(* CODESYS project GenPanel.project

Project tree, tasks and I/O mapping:
  Device : SPK1xx, Production association OWEN, version 3.5.4.26
    application Application
      libraries: Standard, * (System); SysCom, 3.5.5.0 (System); Memory, 3.5.7.0 (3S - Smart Software Solutions GmbH); CmpVisuHandler, 3.5.11.0 (System); SysTypes Interfaces, * (System); VisuDialogs, * (System)
      task MainTask (cyclic, interval t#500ms, priority 1) calls PLC_PRG
      task Task_ReadMercury230 (cyclic, interval t#1ms, priority 20) calls POU_ReadPortGen, POU_VisuDailyEnergies
      task VISU_TASK (cyclic, interval 150 ms, priority 6) calls VisuElems.Visu_Prg
      task Task_DispatchDevices (cyclic, interval t#600ms, priority 20) calls POU_DispatchDevices
      task Task_TraceCurrents (cyclic, interval t#150ms, priority 31) calls POU_TraceCurrents
      task Task_Vis_P (cyclic, interval t#100ms, priority 5) calls POU_TracePowerActive
      task Task_WriteFile (cyclic, interval t#90ms, priority 3) calls POU_File
      task AlarmManagerTask (cyclic, interval 50 ms, priority 0) calls AlarmManager.Alarm_Prg
      program PLC_PRG [ST]
      visualisation Visualization
      visualisation Visualization_DispatchDevices
      visualisation Visualization_DailyEnergies
      visualisation Visualization_P
      global variables GVL
      visualisation Visualization_Energies
      visualisation Visualization_EnergiesDay
      data type FileWork
      visualisation Visualization_ConfigDailyView
      visualisation Visualization_Status
      Alarm Configuration
        alarm class Error (priority 10, acknowledge REP_ACK)
        alarm class Warning (priority 30, acknowledge REP)
        alarm class Info (priority 100, acknowledge REP)
        AlarmStorage
        text list AlarmGroup
        alarm group AlarmGroup
    Buzzer : Buzzer, Production association OWEN, version 3.5.4.0
        unmapped channels: Buzzer enabled, Enable buzzer
    Drives : Drives, Production association OWEN, version 3.5.4.3
        input  Application.fDebugSystem1 : BIT  // Drives info
        output Application.POU_File.fMMCMounted : BIT  // MMC Mounted
        output Application.POU_File.lwMMCSize : LWORD  // MMC size
        output Application.POU_File.lwMMCUsed : LWORD  // MMC used
        output Application.POU_File.lwMMCFree : LWORD  // MMC free
        unmapped channels: FS size, FS used, FS free, USB1 Mounted, USB1 Unmount, USB1 Unmount done, USB1 size, USB1 used, USB1 free, MMC Unmount, MMC Unmount done
    Screen : Screen, Production association OWEN, version 3.5.4.1
        unmapped channels: Get brightness, Dim time, Off time, Full brightness, Dim brightness, Off brightness, Dim visu name, Off visu name, On visu name, Wake up
    Debug : Debug, Production association OWEN, version 3.5.7.10
        input  Application.fDebugSystem : BIT  // Debug info
        input  Application.timeDebugSystem : WORD  // Debug pause
        unmapped channels: RAM used, RAM free, Open files, Processor usage, Core temp
    Modbus_COM : Modbus COM, 3S - Smart Software Solutions GmbH, version 3.4.0.0
        settings: ComPort = 2
      Modbus_Master_COM_Port : Modbus Master, COM Port, 3S - Smart Software Solutions GmbH, version 3.5.5.0
        Modbus_Slave_COM_Port : Modbus Slave, COM Port, 3S - Smart Software Solutions GmbH, version 3.5.4.0
            settings: Channel 0.Function Code = 3; Channel 0.Read Offset = 16#0001; Channel 0.Read Length = 2; Channel 0.Write Offset = 0; Channel 0.Write Length = 0; Channel 0.Cycle Time = 100; Channel 1.Function Code = 3; Channel 1.Read Offset = 16#0003; Channel 1.Read Length = 2; Channel 1.Write Offset = 0; Channel 1.Write Length = 0; Channel 1.Cycle Time = 100; Channel 2.Function Code = 3; Channel 2.Read Offset = 16#0005; Channel 2.Read Length = 2; Channel 2.Write Offset = 0; Channel 2.Write Length = 0; Channel 2.Cycle Time = 100; Channel 3.Function Code = 4; Channel 3.Read Offset = 16#0019; Channel 3.Read Length = 2; Channel 3.Write Offset = 0; Channel 3.Write Length = 0; Channel 3.Cycle Time = 100; Channel 4.Function Code = 3; Channel 4.Read Offset = 16#001B; Channel 4.Read Length = 2; Channel 4.Write Offset = 0; Channel 4.Write Length = 0; Channel 4.Cycle Time = 100; Channel 5.Function Code = 3; Channel 5.Read Offset = 16#001D; Channel 5.Read Length = 2; Channel 5.Write Offset = 0; Channel 5.Write Length = 0; Channel 5.Cycle Time = 100; Channel 6.Function Code = 3; Channel 6.Read Offset = 16#001F; Channel 6.Read Length = 2; Channel 6.Write Offset = 0;
              Channel 6.Write Length = 0; Channel 6.Cycle Time = 100; Channel 7.Function Code = 3; Channel 7.Read Offset = 16#002F; Channel 7.Read Length = 2; Channel 7.Write Offset = 0; Channel 7.Write Length = 0; Channel 7.Cycle Time = 100; Channel 8.Function Code = 3; Channel 8.Read Offset = 16#0037; Channel 8.Read Length = 2; Channel 8.Write Offset = 0; Channel 8.Write Length = 0; Channel 8.Cycle Time = 100; Channel 9.Function Code = 3; Channel 9.Read Offset = 16#00B9; Channel 9.Read Length = 1; Channel 9.Write Offset = 0; Channel 9.Write Length = 0; Channel 9.Cycle Time = 100
            input  Application.IrmsA : ARRAY[0..1] OF WORD  // Channel 0
            input  Application.IrmsB : ARRAY[0..1] OF WORD  // Channel 1
            input  Application.IrmsC : ARRAY[0..1] OF WORD  // Channel 2
            input  Application.P_A : ARRAY[0..1] OF WORD  // Channel 3
            input  Application.P_B : ARRAY[0..1] OF WORD  // Channel 4
            input  Application.P_C : ARRAY[0..1] OF WORD  // Channel 5
            input  Application.P_ABC : ARRAY[0..1] OF WORD  // Channel 6
            input  Application.S_ABC : ARRAY[0..1] OF WORD  // Channel 7
            input  Application.PF_ABCS : ARRAY[0..1] OF WORD  // Channel 8
            unmapped channels: Channel 9
  libraries: VisuSymbols, 3.5.10.0 (System); BASIC, 3.3.3.0 (OSCAT); CAA File, 3.5.3.0 (CAA Technical Workgroup)
  program POU_ReadPortGen [ST]
  program POU_DispatchDevices [ST]
  program POU_TraceCurrents [ST]
  program POU_TracePowerActive [ST]
  program POU_VisuDailyEnergies [ST]
  text list GlobalTextList
  function KAV_HEX_TO_BYTE [ST]
  program POU_File [ST]
  text list System
  image pool ImagePool
  5ce3da45-db07-42e7-a21c-a00fff4ed8f6|D:\A_Kudryashov\Documents\Мои рисунки\setup-clipart-wrench-outline-icon-clip-art_f_85-85.jpg
  Functions/
    function HEXb_TO_byteb [ST]
    function CalcCRC [ST]
    function DWORD_TO_HEXStr [ST]
*)

// Device/Application/FileWork
{attribute 'qualified_only'}
{attribute 'strict'}
TYPE FileWork :
(
	OPEN 			:= 	0,
	CREATE  		:=  10,
	READ			:=	20,
	SET_READ_POS 	:=  30,
	WRITE			:=	40,
	FLUSH			:=	50,
	CLOSE			:= 	60,
	GET_SIZE		:=	70,
	SET_POS			:=	80,
	READ_BLOCK		:=	90
);
END_TYPE

// Device/Application/GVL
VAR_GLOBAL
	IrmsA:REAL;
	IrmsB:REAL;
	IrmsC:REAL;
	Sec:BYTE;
	F_ABCS:REAL;
	PF_ABCS:real; //считанный коэф мощности
	
	P_ABCS_T:REAL;
	
	P_A:REAL; //акивна мощность фазы А
	P_B:REAL; //акивна мощность фазы B
	P_C:REAL; //акивна мощность фазы C
	P_ABC:REAL; // активная мощность
	Pq_ABC:REAL; //актвная мощость в кВт
	S_ABC:REAL; //полная мощность по фазам

	
	StartTrace:BOOL := TRUE;	//Разрешить запуск трассировки
	StopTrace:BOOL	:= FALSE;
	
	MercurySec: BYTE;  //Секунды, считанные из Меркурий230
	MercuryMin: BYTE;
	MercuryHour: BYTE;
	MercuryDay: BYTE;
	MercuryMonth: BYTE;
	MercuryYear: BYTE;
	MercuryEnergyA:DWORD;
	RealDaylyEnergyA:REAL;	//Расчитанная активная энергия за сутки 
	RealDaylyEnergyR:REAL;	//Расчитанная реактивная энергия за сутки
	RealMonthEnergyA:REAL;	//Расчитанная активная энергия за месяц
	RealMonthEnergyR:REAL;  //Расчитанная реактивная энергия за месяц             
	
	fStartTimerOpenSection: BOOL := TRUE; // Старт таймера для открытия сессии
	fStartTimerReadOpenSection:BOOL;
	fStartTimerReadTime:BOOL;
	fStartTimerReadEnergies:BOOL;
	
	DailyEnergies: ARRAY [0..24] OF REAL;
	strDailyEnergies: ARRAY [1..24] OF STRING;
	
	fFirstStartLoadDataFromFile:BOOL := true; //
	
	ReadPosition: DWORD := 5;
	fContinueRead: BOOL := FALSE; // дополнительная переменная, использования при считывании из файла
	
	fDebugSystem:BOOL := TRUE; //разрешить сбор отладочной инфы с панели
	fDebugSystem1:BOOL := TRUE; //разрешить сбор отладочной инфы с панели	
	timeDebugSystem:WORD := 5;
	
	(*
		Переменные для менеджера тревог
	*)
	fLowStorageMem:bool:=false; // используется для фиксации момента, когда на SD-карте останется меньше 20Мб
END_VAR

// Device/Application/PLC_PRG
PROGRAM PLC_PRG
VAR
	
	
END_VAR

VAR_INPUT     
	XCoord:array [0..24] of int; //координаты Х, используемые для расстановки значений мощностей по шкале
    DotY: ARRAY [1..24] OF INT; //координаты часовых точек на графике	
	DotX: ARRAY [1..24] OF INT; // координаты часовых меток на оси Y
	arrMetkaX: ARRAY [1..24] OF STRING := ['01','02','03','04','05','06','07','08','09','10','11','12','13','14','15','16','17','18','19','20','21','22','23','00']; //метки по оси Х
	
	iVar: BYTE := 16#5F;
	CRC:WORD;
	READ_ENERGIES_NOVEMBER:STRING(6) := '$5f$05$3b$00';
	l:byte;
END_VAR

l := 1;
CRC :=MEM.CRC16_Modbus(pMemoryBlock:= adr(READ_ENERGIES_NOVEMBER), uiLength:= 4);

END_PROGRAM

// POU_ReadPortGen
// This example shows how to communicate via the library SysCom.
PROGRAM POU_ReadPortGen
VAR CONSTANT
	n: BYTE := 11;
	TEST_NET: WORD := 16#5F00;
	
	AdrMercury230:string := '$5f'; // адрес текущего счетчика в формате HEX
	PURE_OPEN_CHANEL: STRING(3):= '$05$3b$00'; //команда счетчику на открытие сессии
	READ_ENERGIES_DAYLY:STRING(6) := '$5f$05$4b$00$34$C1'; //чтение потребленных энергий за сутки
	READ_ENERGIES_NOVEMBER:STRING(6) := '$5f$05$3b$00$11$01';
	OPEN_CHANEL: STRING(11) := '$5F$01$02$02$02$02$02$02$02$0D$F4';
	READ_CURRENT_TIME : STRING(6) := '$5F$04$00$43$12';	
	strHex:STRING(3) := '16#';
END_VAR
VAR
	bOpenCom: BOOL := TRUE;
	hCom: RTS_IEC_HANDLE := RTS_INVALID_HANDLE;
	Result: RTS_IEC_RESULT;
	csComSettings: COM_Settings;
	bWriteCom: BOOL := TRUE;
	dwWritten: UDINT;
	dwOffset: UDINT;
	str : STRING := '$5F$01$02$02$02$02$02$02$02$0D$F4';
	strTempCRC:STRING;
	strTempCRC20:STRING(20);
	abyWriteData: ARRAY[0..n-1] OF BYTE;
	i, xxx: INT;
	bReadCom: BOOL := TRUE;
	dwRead: UDINT;
	strRead: STRING(30);
	dwWrittenLog : ARRAY[0..49] OF DWORD;
	dwZeroWrittenCount : DWORD;
	iCurWrittenLog : INT;
	myCRC: DWORD := 0;
	myData: DWORD := 0;
	myPTR: POINTER TO STRING;
	length:INT;
	TimeOut, TimeOut1:TP;
	TimerDelayOpenSection, TimerDelayReadSection, TimerDelayReadEnergies:TON;
	TimerDelayReadTime:TON;
	myElapsedTime: TIME := t#0ms;
	
	varTime: TIME := T#0S;
	BufferWrite, BufferWriteTime:POINTER TO BYTE;
	BufferRead:POINTER TO BYTE;
	fStartPOU:BOOL := FALSE;
	bufsize:UINT;
	SysError:UDINT;
	strReadSec:string(5);
	strReadEnergy: STRING(4);
	a: INT;
	strForHex: STRING(5);
END_VAR
VAR_INPUT
	TimerBool:bool;
END_VAR

(*
//myData := OPEN_CHANEL;
myPTR := ADR(OPEN_CHANEL);
myCRC := MEM.CRC16_standard(myPTR,2);
*)

strTempCRC := '';
strTempCRC := Concat(STR1:= AdrMercury230, STR2 := PURE_OPEN_CHANEL );//PURE_OPEN_CHANEL
i:= Len(strTempCRC);
myCRC := mem.CRC16_Modbus(ADR(strTempCRC), i+1);
//strTempCRC20 := DWORD_TO_STRING(myCRC);

strTempCRC := Concat(strTempCRC, DWORD_TO_HEXStr(In:= myCRC));


IF bOpenCom THEN
	bOpenCom := FALSE;
	// Prepare test data

	// Open COM port 1
	hCom := SysComOpen(sPort:= SYS_COMPORT3 , pResult:= ADR(Result));
	IF hCom <> RTS_INVALID_HANDLE THEN
		// Configure the connection
		csComSettings.byParity := SYS_NOPARITY;
		csComSettings.byStopBits := SYS_ONESTOPBIT;
		csComSettings.sPort := SYS_COMPORT3;
		csComSettings.ulBaudrate := SYS_BR_9600;
		csComSettings.ulBufferSize := 0;
		csComSettings.ulTimeout := 10;
		Result := SysComSetSettings(hCom:= hCom, pSettings:= ADR(csComSettings) , pSettingsEx:= 0);
	END_IF
	
	SysComSetTimeout(hCom:= hCom, ulTimeout := 200);
END_IF

{
//Тест на открытие канал общения между счетчиком и панелью
length := SIZEOF(OPEN_CHANEL);
length := 11;

FOR i:=0 TO (length-1) DO
	abyWriteData[i] := 0;	
END_FOR

FOR i:=0 TO (length-1) DO
	abyWriteData[i] := OPEN_CHANEL[i MOD (length)];
END_FOR
	
IF hCom <> RTS_INVALID_HANDLE THEN
	// Write data
	dwWritten := SysComWrite(hCom:= hCom,	pbyBuffer:= ADR(abyWriteData)+dwOffset,	ulSize:= SIZEOF(abyWriteData)-dwOffset,	ulTimeout:= 100,	pResult:= ADR(Result) );
	IF dwWritten = 0 THEN
		dwZeroWrittenCount := dwZeroWrittenCount + 1;
	ELSE
		dwWrittenLog[iCurWrittenLog] := dwWritten;
		iCurWrittenLog := iCurWrittenLog + 1;
		IF iCurWrittenLog > 49 THEN
			iCurWrittenLog := 0;
		END_IF
	END_IF
	dwOffset := dwOffset + dwWritten;
	IF dwOffset >= SIZEOF(abyWriteData) THEN
		bWriteCom := FALSE;
		dwOffset := 0;
	END_IF
END_IF

TimeOut(IN:=TRUE,PT:=T#150MS);
IF TimeOut.Q THEN
	IF hCom <> RTS_INVALID_HANDLE AND bReadCom THEN
		// Read data
		dwRead := SysComRead(hCom:= hCom,	pbyBuffer:= ADR(strRead),	ulSize:= SIZEOF(strRead),	ulTimeout:= 5000,	pResult:= ADR(Result));
	
	END_IF
END_IF
*}
	
//Реализовать проверку на наличие канала

//Проверка на открытую сессию

//TimerDelayOpenSection(IN:=GVL.fStartTimerOpenSection, PT := T#20S);
//IF TimerDelayOpenSection.Q THEN
	//Открытие канала
	
	IF (hCom <> RTS_INVALID_HANDLE) AND NOT fStartTimerReadOpenSection THEN
		// Write data
		dwWritten := SysComWrite(hCom:= hCom,	pbyBuffer:= ADR(strTempCRC(*OPEN_CHANEL*)),	ulSize:= 11*SIZEOF(BYTE),	ulTimeout:= 200,	pResult:= ADR(Result) );
		(*IF dwWritten = 0 THEN
		dwZeroWrittenCount := dwZeroWrittenCount + 1;
	ELSE
		dwWrittenLog[iCurWrittenLog] := dwWritten;
		iCurWrittenLog := iCurWrittenLog + 1;
		IF iCurWrittenLog > 49 THEN
			iCurWrittenLog := 0;
		END_IF
	END_IF
	dwOffset := dwOffset + dwWritten;
	IF dwOffset >= SIZEOF(abyWriteData) THEN
		bWriteCom := FALSE;
		dwOffset := 0
	END_IF*)
	END_IF
	
	WHILE NOT TimerDelayReadSection.Q DO
		TimerDelayReadSection(In:= TRUE, PT:=T#200MS);
	END_WHILE		
		
	TimerDelayReadSection(In:= FALSE, PT:=T#200MS);
	
	
	IF hCom <> RTS_INVALID_HANDLE AND bReadCom THEN
			// Read data			
				dwRead := SysComRead(hCom:= hCom,	pbyBuffer:= ADR(strRead),	ulSize:= 5*SIZEOF(BYTE),	ulTimeout:= 200,	pResult:= ADR(Result));
				gvl.fStartTimerReadOpenSection := FALSE;
	END_IF
	
	
//END_IF

IF NOT TimerDelayOpenSection.Q THEN
	GVL.fStartTimerOpenSection := true;
END_IF

//Чтение текущего времени

length := n;

	
IF (hCom <> RTS_INVALID_HANDLE) THEN
	//Очистим буфер FIFO
	SysError := SysComPurge(hCom:= hCom);
	// Write data
	dwWritten := SysComWrite(hCom:= hCom,	pbyBuffer:= ADR(READ_CURRENT_TIME),	ulSize:= 5*SIZEOF(BYTE),	ulTimeout:= 200,	pResult:= ADR(Result) );
END_IF

	
gvl.fStartTimerReadTime := TRUE;
WHILE NOT TimerDelayReadTime.Q DO 
	TimerDelayReadTime(IN:=gvl.fStartTimerReadTime, PT:=T#200MS);
END_WHILE
//IF TimerDelayReadTime.Q THEN
	IF hCom <> RTS_INVALID_HANDLE AND bReadCom THEN
		bufsize := SIZEOF(strRead)-1;
		dwRead := SysComRead(hCom:= hCom,	pbyBuffer:= ADR(strRead),	ulSize:= 11,	ulTimeout:= 200,	pResult:= ADR(Result));
	
		bOpenCom := FALSE;
		IF dwRead > 5 THEN
			
			GVL.MercurySec:= HEXb_TO_byteb(strRead[1]);
			GVL.MercuryMin:= HEXb_TO_byteb(strRead[2]);
			GVL.MercuryHour:= HEXb_TO_byteb(strRead[3]);
			GVL.MercuryDay:= HEXb_TO_byteb(strRead[5]);
			GVL.MercuryMonth:= HEXb_TO_byteb(strRead[6]);
			GVL.MercuryYear:= HEXb_TO_byteb(strRead[7]);
			
			//OSCAT_BASIC._STRING_TO_BUFFER(STR:=strRead , POS:=3 , PT:=ADR(strForHex) , SIZE:= 1);
			//strForHex:='16#';
			
			//strForHex := OSCAT_BASIC.BUFFER_TO_STRING(PT:= ADR(strRead) , SIZE:=30 , START:=3 , STOP:=3 );
			//strForHex:= CONCAT(strHex,strForHex );
			//strForHex := strForHex + '16#'; 
			//insert(strForHex,strhex,2);
			//a := OSCAT_BASIC.FSTRING_TO_BYTE(IN:=strForHex);
			//strForHex := OSCAT_BASIC.CHR_TO_STRING(C:=strRead[3]);
			//a:=  OSCAT_BASIC.DEC_TO_BYTE(DEC:=strForHex);
			//a:= OSCAT_BASIC.CODE(strRead,4);
			//a:=KAV_HEX_TO_BYTE(strForHex);
		END_IF	
		
	TimerDelayReadTime(IN:=FALSE, PT:=T#200MS);
	MEM.MemFill(pMemoryBlock:= ADR(strRead), uiLength:= 30*SIZEOF(BYTE), byFillValue:= 0);
	
	END_IF	
//END_IF	
	
	
//---Чтение энергий
//---Энергии за сутки
IF (hCom <> RTS_INVALID_HANDLE) THEN
	// Write data
	dwWritten := SysComWrite(hCom:= hCom,	pbyBuffer:= ADR(READ_ENERGIES_DAYLY),	ulSize:= 6*SIZEOF(BYTE),	ulTimeout:= 200,	pResult:= ADR(Result) );
END_IF

WHILE NOT TimerDelayReadEnergies.Q DO 
	TimerDelayReadEnergies(IN:=TRUE, PT:=T#290MS);
END_WHILE

	IF hCom <> RTS_INVALID_HANDLE AND bReadCom THEN
		// Read data
		//MEM.MemFill(pMemoryBlock:= ADR(strRead), uiLength:= 30*SIZEOF(BYTE), byFillValue:= 0);
		dwRead := SysComRead(hCom:= hCom,	pbyBuffer:= ADR(strRead),	ulSize:= SIZEOF(strRead),	ulTimeout:= 400,	pResult:= ADR(Result));
		
		bOpenCom := FALSE;
			
		MercuryEnergyA := strRead[2];	
		MercuryEnergyA := SHL(MercuryEnergyA,8);
		MercuryEnergyA := MercuryEnergyA + strRead[1];
		MercuryEnergyA := SHL(MercuryEnergyA,8);
		MercuryEnergyA := MercuryEnergyA + strRead[4];
		MercuryEnergyA := SHL(MercuryEnergyA,8);
		MercuryEnergyA := MercuryEnergyA + strRead[3];
		
		gvl.RealDaylyEnergyA := OSCAT_BASIC.ROUND(in:= (MercuryEnergyA / 100.0), N := 2); //      /1000  * 10(коэф трасформации)
			
		//GVL.MercuryHour := 00;
		
		FOR i:= GVL.MercuryHour TO INT_TO_BYTE(SIZEOF((gvl.DailyEnergies))/SIZEOF(REAL))-1 BY 1 DO
			gvl.DailyEnergies[i] := 0;
		END_FOR
		
		gvl.DailyEnergies[GVL.MercuryHour] := gvl.RealDaylyEnergyA;
		
	END_IF

TimerDelayReadEnergies(IN:=FALSE, PT:=T#290MS);

//Энергии за месяц текущий

IF (hCom <> RTS_INVALID_HANDLE) THEN
	// Write data
	dwWritten := SysComWrite(hCom:= hCom,	pbyBuffer:= ADR(READ_ENERGIES_NOVEMBER),	ulSize:= 6*SIZEOF(BYTE),	ulTimeout:= 200,	pResult:= ADR(Result) );
END_IF

WHILE NOT TimerDelayReadEnergies.Q DO 
	TimerDelayReadEnergies(IN:=TRUE, PT:=T#290MS);
END_WHILE

	IF hCom <> RTS_INVALID_HANDLE AND bReadCom THEN
		// Read data
		MEM.MemFill(pMemoryBlock:= ADR(strRead), uiLength:= 30*SIZEOF(BYTE), byFillValue:= 0);
		dwRead := SysComRead(hCom:= hCom,	pbyBuffer:= ADR(strRead),	ulSize:= SIZEOF(strRead),	ulTimeout:= 400,	pResult:= ADR(Result));
		
		MercuryEnergyA := 0;
		
		bOpenCom := FALSE;
			
		MercuryEnergyA := strRead[2];	
		MercuryEnergyA := SHL(MercuryEnergyA,8);
		MercuryEnergyA := MercuryEnergyA + strRead[1];
		MercuryEnergyA := SHL(MercuryEnergyA,8);
		MercuryEnergyA := MercuryEnergyA + strRead[4];
		MercuryEnergyA := SHL(MercuryEnergyA,8);
		MercuryEnergyA := MercuryEnergyA + strRead[3];
		
		gvl.RealMonthEnergyA := (MercuryEnergyA / 100.0);
		
		
	END_IF

TimerDelayReadEnergies(IN:=FALSE, PT:=T#290MS);

IF NOT bOpenCom THEN
	hCom := SysComClose(hCom:= hCom);
	IF hCom <> RTS_INVALID_HANDLE  THEN
		bOpenCom := TRUE;
	END_IF
END_IF

END_PROGRAM

// Functions/DWORD_TO_HEXStr
//Функция конвертирует значение DWORD в строку, которая содержит значения в виде HEX
FUNCTION DWORD_TO_HEXStr : STRING(4)
VAR_INPUT
	In:DWORD;
END_VAR
VAR
	AdrValue:POINTER TO BYTE;
	TempStr:STRING(4) := '';
	//i:=BYTE := 0;
	i: INT := 0;
END_VAR

AdrValue := ADR(In);

FOR i:=0 TO 4-1 DO
	DWORD_TO_HEXStr[i] := (AdrValue^);
	AdrVAlue := AdrVAlue +1;
END_FOR

END_FUNCTION

// Functions/HEXb_TO_byteb
// Функция принимает hex-значение в byte и выдает DEC в типе byte
FUNCTION HEXb_TO_byteb : BYTE
VAR_INPUT
	In:BYTE;
END_VAR
VAR
END_VAR

	IF In <= 16#9 THEN
		HEXb_TO_byteb := In;		
	ELSIF In >= 16#10 AND In <=16#19 THEN
		HEXb_TO_byteb :=  In - 6;		
	ELSIF In>=16#20 AND In<=16#29 THEN
		HEXb_TO_byteb :=  In - 12;		
	ELSIF In >= 16#30 AND In <=16#39 THEN
		HEXb_TO_byteb :=  In - 18;	
	ELSIF In >=16#40 AND In <= 16#49 THEN
		HEXb_TO_byteb :=  In - 24;
	ELSIF In >= 16#50 AND In <= 16#59 THEN
		HEXb_TO_byteb :=  In - 30;	
	ELSE
		HEXb_TO_byteb := In;
	END_IF;

END_FUNCTION

// KAV_HEX_TO_BYTE
FUNCTION KAV_HEX_TO_BYTE : BYTE
VAR_INPUT
	HEX : STRING(5);
END_VAR
VAR
	pt : POINTER TO BYTE;
	i: INT;
	X: BYTE;
	stop: INT;
	//KAV_HEX_TO_BYTE:BYTE;
END_VAR

(*
pt := ADR(hex);
stop := LEN(hex);
FOR I := 1 TO stop DO
	(* read the first character and subtract 48 to get value in decimal 0 = 48 *)
	x := pt^;
	(* calculate the value of the digit *)
	IF X > 47 AND x < 58 THEN
		KAV_HEX_TO_BYTE := SHL(KAV_HEX_TO_BYTE,4) + X - 48;
		pt := pt + 1;
	ELSIF X > 64 AND X < 71 THEN
		KAV_HEX_TO_BYTE := SHL(KAV_HEX_TO_BYTE,4) + X - 55;
		pt := pt + 1;
	ELSIF X > 96 AND X < 103 THEN
		KAV_HEX_TO_BYTE := SHL(KAV_HEX_TO_BYTE,4) + X - 87;
		pt := pt + 1;
	ELSe
		KAV_HEX_TO_BYTE := pt^;
	END_IF;
	
END_FOR;
*)

pt := ADR(hex);
stop := LEN(hex);
FOR I := 1 TO stop DO
	(* read the first character and subtract 48 to get value in decimal 0 = 48 *)
	x := pt^;
	(* calculate the value of the digit *)
	IF x <= 9 THEN
		KAV_HEX_TO_BYTE := x;
		pt := pt + 1;
	ELSIF X > 9 AND X <=19 THEN
		KAV_HEX_TO_BYTE :=  X - 6;
		pt := pt + 1;	
	ELSIF x>19 AND x<24 THEN
		KAV_HEX_TO_BYTE :=  X - 12;
		pt := pt + 1;		
	ELSE
		KAV_HEX_TO_BYTE := pt^;
	END_IF;
	
END_FOR;

END_FUNCTION

// POU_VisuDailyEnergies
PROGRAM POU_VisuDailyEnergies
VAR
	arrPolylineCoord: ARRAY [0..24] OF VisuStructPoint;
	iPolylinePoints: INT := 24;
	iIndex:INT := 1;
	MaxValueDailyEnergies:REAL;
	scale:REAL:=0; //масштабный коэф
	i:BYTE;
	Count:byte:=0;
	//DailyEnergiesTemp: array [0..24] of real := [8,1,2,3,4,5,6,7,8,9,10,11,12,13,14,15,16,17,18,19,20,21,22,23,8];
END_VAR

VAR CONSTANT
	XAxysX0 : WORD := 10;  //начальная координата Х нулевой оси
	XAxysX1 : WORD := 795; //конечная координата Х нулевой оси
	XAxysStep : WORD := ((XAxysX1 - XAxysX0) / 25) + 1; 
	XAxysY0 : WORD := 400;
	AAxysY1 : WORD := 400; 
	YAxysX0 : WORD := 5;
	YAxysX1 : WORD := 5;
	YAxysY0 : WORD := 110;
	YAxysY1 : WORD := 410;
	YAxysStep : WORD := ((YAxysY1 - YAxysY0 -10) / 24);
END_VAR

VAR_INPUT
	DailyViewConfig:BYTE := 0; //от этого значения будет зависеть что график будет отображать: показания на текущуб дату или на выбранную
	Calender:DATE; 
END_VAR

(*
Но вот, на всякий случай, вариант "классической нормировки":

Пусть требуется ряд значений {X1, X2 ... Xn} или далеее {Xi}, i = 1..n, 
промасштабировать в интервал [A,B] и получить новые значения {X'i}, 
так чтобы минимум ряда (Xmin) преобразовался в значение A, а максимум (Xmax) в B:

 Имеем Xmin <= Xi <= Xmax для любого i, будем получать A <= X'i <= B:

scale = (B - A) / (Xmax - Xmin) масштабный множитель
X'i = A + (Xi - Xmin) * scale, для всех i = 1.. n 

*)

iIndex := gvl.MercuryHour;

MaxValueDailyEnergies := OSCAT_BASIC.ARRAY_MAX(pt:= ADR((*gvl.DailyEnergies*)gvl.DailyEnergies), size:= 24*SIZEOF(REAL));
IF  MaxValueDailyEnergies = 0 THEN
	MaxValueDailyEnergies := 1;
END_IF


scale := ((YAxysY1 - YAxysY0) / (MaxValueDailyEnergies - 0));
Count := INT_TO_BYTE( SIZEOF(arrPolylineCoord) / SIZEOF(VisuStructPoint));
FOR i:=0 TO Count-1 BY 1 DO
	arrPolylineCoord[i].iX := (i)* XAxysStep + XAxysX0; //Номер часа
	arrPolylineCoord[i].iY := TRUNC_INT(YAxysY1 - (gvl.DailyEnergies[i] - 0)* scale);
	
	plc_prg.XCoord[i] := arrPolylineCoord[i].iX;
	//для установки точки на графике
	IF i>0 THEN
		//т.к. точек графика меньше кол-ва 
		plc_prg.DotY[i] := - (YAxysY1 - arrPolylineCoord[i].iY);
		plc_prg.DotX[i] := arrPolylineCoord[i].iX;  // - 3    - учитывается ширина точки 
	END_IF
	
END_FOR

END_PROGRAM

// POU_DispatchDevices
PROGRAM POU_DispatchDevices
VAR
	DispVar:UINT;	// переменная, в которой хранится считанное значение состояний входов модуля ввода
	DispContactor:BOOL; //контактор вклл/выкл
	tempContactor:UINT;
	DispUPP:BOOL;	//устройство плавного пуска вкл/выкл
	DispFreqInverter:BOOL;	//ЧРП вкл/выкл
END_VAR


IF DispVar = 1 THEN
	DispContactor := TRUE;
	ELSE
		DispContactor := FALSE;	
END_IF

IF DispVar = 2 THEN
	DispUPP := TRUE;
	ELSE
		DispUPP := FALSE;	
END_IF

IF DispVar = 4 THEN
	DispFreqInverter := TRUE;
	ELSE
		DispFreqInverter := FALSE;	
END_IF

END_PROGRAM

// POU_TraceCurrents
PROGRAM POU_TraceCurrents
VAR
		TraceIrmsA:REAL;
	TraceIrmsB:REAL;
	TraceIrmsC:REAL;
END_VAR

	TraceIrmsA:=IrmsA;
	TraceIrmsB:=IrmsB;
	TraceIrmsC:=IrmsC;

END_PROGRAM

// POU_TracePowerActive
PROGRAM POU_TracePowerActive
VAR
	TraceAPowerA:REAL;
	TraceAPowerB:REAL;
	TraceAPowerC:REAL;
	TraceAPowerABC:REAL;
	
	TraceSPowerABC:REAL;
	
	PowerCounter_TOF:TOF;
END_VAR

VAR RETAIN
	CounterPower:LREAL;
END_VAR

	TraceAPowerA := ABS(P_A / 1000);
	TraceAPowerB := ABS(P_B / 1000);
	TraceAPowerC := ABS(P_C / 1000);
	
	TraceAPowerABC := ABS(P_ABC / 1000);
	
	TraceSPowerABC := ABS( S_ABC / 1000) ;
	
	PowerCounter_TOF(IN := TRUE, PT:= T#1S); 
	
	IF PowerCounter_TOF.Q THEN
		//POU_PowerCounter.fStartTimer:=TRUE;
		
		CounterPower := (TraceSPowerABC / 3600) + CounterPower;
		
		ELSE
			//POU_PowerCounter.fStartTimer:=FALSE;
		
	END_IF

END_PROGRAM

// POU_File
PROGRAM POU_File
VAR
	hFile:	FILE.CAA.HANDLE;					// дескриптор открытого файла; // дескриптор файла
	
	fMMCMounted:BOOL; // флаг смонтированного носителя
	lwMMCSize:LWORD; // размер карты памяти
	lwMMCUsed:LWORD; // кол-во занятой памяти
	lwMMCFree:LWORD; // кол-во свободной памяти
	i:DINT;
	fbFileOpen:      FILE.Open;
    fbFileWrite:      FILE.Write;
    fbFileRead:      FILE.Read;
	fbFileReadBlock:		FILE.Read;
    fbFileClose:      FILE.Close;
	fbFileFlush:					FILE.Flush;							// ФБ сброса буфера в файл
	fbFileGetSize:					FILE.GetSize;						// ФБ получения размера файла
	fbFileSetPos:		File.SetPos;
	fbFileEOF:			File.EOF;
	// // шаг операции с файлом
	eState: FileWork := FileWork.GET_SIZE; // индикатор позиции при записи из файла
	
	eStateReadFile: FileWork := FileWork.OPEN;
	
	sFileName: STRING;
	xWBusy: BOOL;
	udiArchSize:					UDINT;								// размер архива в байтах	
	//strTemp:STRING; := '0';
	strTemp: STRING(255) := '';
	timerOn:TON;
	Count:UDINT := 0;
	FileSize : UdINT; //размер файла для чтения
	TimerWriteToFile: TON;
	TimerDelay: TON;
	// Флаг устанавливается, когда найден интересующий блок данных
	fFindBlock: BOOL := FALSE;
	
	strExceptionText : STRING;
	exc : __SYSTEM.ExceptionCode;
	// Переменная для формирования числа
	TempStrDigit: STRING := '';
	// Используется для подсчета количества дневных значений
	n: WORD := 0;
	BlockBuffer: ARRAY [0..255] OF STRING;
	ptrBlockBuffer:POINTER TO STRING;
	index:UINT := 0;
END_VAR

VAR CONSTANT
	csDir : STRING := '/mnt/ufs/media/mmcblk0p1/'; //каталог хранения файлов
	csDaily: STRING := 'daily.csv'; //храним суточные данные
	csMonths: STRING := 'months.csv'; // храним месячные данные
	csYears : STRING := 'years.csv';  // храним годовые данные
	TimePeriod:TIME := T#10M;
	
	MARKER_DATA :STRING := '#data';
END_VAR

IF (gvl.MercuryDay > 0) OR (gvl.MercuryMonth>0) OR (gvl.MercuryYear > 0) THEN
// сформируем имя файла на основе текущей даты
sFileName	:=	CONCAT(csDir, BYTE_TO_STRING(gvl.MercuryDay));
sFileName := concat(sFileName, '_');
sFileName	:=	concat(sFileName, BYTE_TO_STRING(gvl.MercuryMonth));
sFileName := concat(sFileName, '_'); 
sFileName	:=	concat(sFileName, BYTE_TO_STRING(gvl.MercuryYear));
sFileName := concat(sFileName, '.csv'); 

//Проверим смонтированна ли карта памяти. ДА - пишем на нее, Нет - не пишем
IF fMMCMounted THEN
	IF NOT gvl.fFirstStartLoadDataFromFile THEN
		IF (lwMMCUsed <= (lwMMCSize - 16#1312D00)) then //Если на карте памяти осталось не меньше 20МБ
	
		//сделаем периодичность
		//в 10сек
	
			IF NOT TimerWriteToFile.Q THEN
				TimerWriteToFile(In:= TRUE, pt := TimePeriod);
			END_IF
	
			IF TimerWriteToFile.ET = TimePeriod THEN

				CASE eState OF
	
					FileWork.OPEN:	// шаг открытия файла

				
						fbFileOpen(xExecute:=TRUE, sFileName:=sFileName, eFileMode:=FILE.MODE.MAPPD);	
			
			
						// если файл, в который производится запись, не существует, то создадим его и запишем в него заголовок архива
						IF fbFileOpen.eError=FILE.ERROR.NOT_EXIST THEN
							fbFileOpen(xExecute:=FALSE);
							eState	:=	FileWork.CREATE;
						END_IF
	
						// если файл существует и был успешно открыт, то переходим к шагу записи в файл
						IF fbFileOpen.xDone THEN
							hFile	:=	fbFileOpen.hFile;
							fbFileOpen(xExecute:=FALSE);
	
							eState	:=	FileWork.WRITE;
						END_IF
		
			
					FileWork.CREATE:	// шаг создания файла	
	
						// в созданном файле еще нет записей
						//uiArchEntry:=0;
	
						fbFileOpen(xExecute:=TRUE, sFileName:=sFileName, eFileMode:=FILE.MODE.MWRITE);
	
						IF fbFileOpen.xDone THEN
							hFile	:=	fbFileOpen.hFile;
							fbFileOpen(xExecute:=FALSE);
				
								// после создания файла можно перейти к шагу записи данных
							eState	:=	FileWork.WRITE;
						END_IF	
			
						IF fbFileOpen.xError THEN
							// обработка ошибок
						END_IF
	
	
					FileWork.WRITE:	// шаг записи в буфер
						//добавим время
						//добавим маркер вставки даты и времени 
						strTemp := '##date';
						strTemp := concat(strTemp,INT_TO_STRING( gvl.MercuryYear));
						strTemp := concat(strTemp, '.');
						strTemp := concat(strTemp, INT_TO_STRING(gvl.MercuryMonth));
						strTemp := concat(strTemp, '.');
						strTemp := concat(strTemp, INT_TO_STRING(gvl.MercuryDay));
						strTemp := concat(strTemp, '.');
						strTemp := concat(strTemp, INT_TO_STRING((gvl.MercuryHour)));
						strTemp := concat(strTemp, '.');
						strTemp := concat(strTemp, INT_TO_STRING((gvl.MercuryMin)));
						strTemp := concat(strTemp, '.');
						strTemp := concat(strTemp, INT_TO_STRING(( gvl.MercurySec)));
						//вставим маркер данных
						strTemp := concat(strTemp, '#data');
				
						Count := SIZEOF(gvl.DailyEnergies) / SIZEOF(REAL);
						FOR i:=0 TO Count-1 BY 1 DO
							strTemp := concat(strTemp, REAL_TO_STRING(gvl.DailyEnergies[i]));
							strTemp := concat(strTemp, '$3B');
						END_FOR
						//Добавим символ переноса строки		
						strTemp := concat(strTemp, '$0D');
					// запись строки архива в файл
						fbFileWrite(xExecute:=TRUE, hFile:=hFile, pBuffer:=ADR(strTemp), szSize:=INT_TO_UDINT(LEN(strTemp)));
					
						strTemp := '';
					
						IF fbFileWrite.xDone THEN
							fbFileWrite(xExecute:=FALSE);
				
						// после записи число строк в архиве увеличилось на одну
						//uiArchEntry:=uiArchEntry+1;
						
						// теперь можно перейти к шагу сброса буфера в файл
							eState	:=	FileWork.FLUSH;
										
						END_IF
			
						IF fbFileWrite.xError THEN
							// обработка ошибок
						END_IF

			
					FileWork.FLUSH: // шаг сброса буфера в файл
			
						fbFileFlush(xExecute:=TRUE, hFile:=hFile);
			
						IF fbFileFlush.xDone THEN
							fbFileFlush(xExecute:=FALSE);
						
						// теперь можно перейти к шагу закрытия файла
							eState:=FileWork.CLOSE;
						END_IF
					
						IF fbFileFlush.xError THEN
						// обработка ошибок
						END_IF
		
			
					FileWork.CLOSE:	// шаг закрытия файла
			
					fbFileClose(xExecute:=TRUE, hFile:=hFile);
			
					IF fbFileClose.xDone THEN
						fbFileClose(xExecute:=FALSE);
						xWBusy	:=	FALSE;				
					
						// теперь можно перейти к шагу определения размера файла
						eState	:=	FileWork.GET_SIZE;
					END_IF
					
					TimerWriteToFile(In:= FALSE, pt := TimePeriod);
					
					FileWork.GET_SIZE:	// шаг определения размера файла
			
					fbFileGetSize(xExecute:=TRUE, sFileName:=sFileName);
						
						// определяем размер файла
						IF fbFileGetSize.xDone THEN
							udiArchSize:=fbFileGetSize.szSize;
							fbFileGetSize(xExecute:=FALSE);
							
							// вернемся на шаг открытия файла для ожидания следующего управляющего сигнала	
							eState	:=	FileWork.OPEN;
						END_IF
						
					// размер несуществующего файла...	
					IF fbFileGetSize.eError=FILE.ERROR.NOT_EXIST THEN
						
						// очевидно, можно интерпретировать как ноль
						udiArchSize	:=	0;
						fbFileGetSize(xExecute:=FALSE);
						
						// вернемся на шаг открытия файла для ожидания следующего управляющего сигнала
						eState			:=	FileWork.OPEN;
					ELSIF  fbFileGetSize.xError THEN
						fbFileGetSize(xExecute:=FALSE);
						eState			:=	FileWork.OPEN;	
					END_IF
					
					
			//установка позиции
						FileWork.SET_POS:
							fbFileSetPos(xExecute := TRUE, hFile := hFile, udiPos := 0);
					
							IF fbFileSetPos.xDone THEN
								eState := FileWork.WRITE;
							END_IF														
						
	
				END_CASE
			END_IF	
		END_IF
	END_IF


	//При первом старте считаем данные из сохранненого файла
	IF gvl.fFirstStartLoadDataFromFile THEN
		CASE eStateReadFile OF
	
			FileWork.OPEN:	// шаг открытия файла

			// if gvl.fContinueRead and TimerDelay.Q then	
				fbFileOpen(xExecute:=TRUE, sFileName:=sFileName, eFileMode:=FILE.MODE.MREAD, xExclusive := true);			
	
			// если файл существует и был успешно открыт, то переходим к шагу чтения из файла
				IF fbFileOpen.xDone THEN
					hFile	:=	fbFileOpen.hFile;
					fbFileOpen(xExecute:=FALSE);
	
					eStateReadFile	:=	FileWork.GET_SIZE;
				
					IF NOT gvl.fContinueRead THEN
						ReadPosition := 5;
					END_IF	
				END_IF
			
				IF fbFileOpen.eError = FILE.ERROR.NOT_EXIST THEN
					eStateReadFile:=FileWork.CLOSE;
					gvl.fFirstStartLoadDataFromFile := false;
				END_IF
	
			FileWork.Read:	
	
				fbFileRead(xExecute:=TRUE, hFile:=hFile, pBuffer:=ADR(strTemp), szBuffer:=LEN(MARKER_DATA));			
			
				IF fbFileRead.xDone THEN
					fbFileRead(xExecute:=FALSE);
		
				// после записи число строк в архиве увеличилось на одну
				//uiArchEntry:=uiArchEntry+1;
					IF OSCAT_BASIC.BUFFER_SEARCH(
												PT:= ADR(strTemp), 
												SIZE:= LEN(strTemp), 
												STR:= MARKER_DATA, 
												POS:= 0, 
												IGN:= FALSE) <> 0 THEN
						ReadPosition := ReadPosition +1;
					
						eStateReadFile := FileWork.SET_POS;
						
						fFindBlock := FALSE;
					ELSe
					
					//Читаем содержимое
					
					//Расчитаем смещение позиции чтения файла
						ReadPosition := (*udiArchSize-(udiArchSize-1)- *)(ReadPosition) - LEN(MARKER_DATA);
					
						fFindBlock := TRUE;
						
						eStateReadFile := FileWork.SET_POS;
					
						strTemp := '';
						ptrBlockBuffer := ADR('');
					
					END_IF
				END_IF
			
			IF fbFileWrite.xError THEN
				// обработка ошибок
			END_IF			
	
			FileWork.CLOSE:	// шаг закрытия файла
	
				fbFileClose(xExecute:=TRUE, hFile:=hFile);
	
				IF fbFileClose.xDone THEN
					fbFileClose(xExecute:=FALSE);
					xWBusy	:=	FALSE;				
				
					gvl.fFirstStartLoadDataFromFile := FALSE;
					IF fFindBlock THEN
						gvl.fFirstStartLoadDataFromFile := FALSE;	
					END_IF	
				END_IF
			
			
			FileWork.GET_SIZE:	// шаг определения размера файла
	
				fbFileGetSize(xExecute:=TRUE, sFileName:=sFileName);
				
				// определяем размер файла
				IF fbFileGetSize.xDone THEN
					udiArchSize:=fbFileGetSize.szSize;
					fbFileGetSize(xExecute:=FALSE);
					
					// вернемся на шаг открытия файла для ожидания следующего управляющего сигнала	
					eStateReadFile	:=	FileWork.SET_POS;
				END_IF
				
			// размер несуществующего файла...	
				IF fbFileGetSize.eError=FILE.ERROR.NOT_EXIST THEN
				
				// очевидно, можно интерпретировать как ноль
					udiArchSize	:=	0;
					fbFileGetSize(xExecute:=FALSE);
				
				// вернемся на шаг открытия файла для ожидания следующего управляющего сигнала
					eState			:=	FileWork.OPEN;
				ELSIF  fbFileGetSize.xError THEN
					fbFileGetSize(xExecute:=FALSE);
					eState			:=	FileWork.READ;	
				END_IF
			
			
	//установка позиции
			FileWork.SET_POS:
				fbFileSetPos(xExecute := TRUE, hFile := hFile, udiPos :=udiArchSize - ReadPosition);							
			
				IF fbFileSetPos.xDone THEN	
					eStateReadFile := FileWork.READ;
					fbFileSetPos(xExecute:= FALSE);
				
					IF fFindBlock THEN
						eStateReadFile := FileWork.READ_BLOCK;
					END_IF		
				END_IF
			
			FileWork.READ_BLOCK: //извлечение данных из блока
				//Очистим бувер, чтобы не было мусора
				//strTemp := '';
				//читает от высчитанной позиции и до конца файла
				fbFileRead(xExecute:=TRUE, hFile:=hFile, pBuffer:=ADR(strTemp), szBuffer:=((ReadPosition)*SIZEOF(BYTE))(*Последний символ "СК" или hex=0D. Он нам не нужен*));
				IF fbFileRead.xDone THEN
					fbFileRead(xExecute := FALSE);
					
					TempStrDigit := '';
					index := 0;
					n:= 0; // индекс массива
					Count := LEN(strTemp);
					FOR i:=0 TO Count-1 BY 1 DO					
						//сравниваем символы до ;
						IF OSCAT_BASIC.BUFFER_SEARCH(
													PT:= ADR(strTemp[i]), 
												SIZE:= 1, 
												STR:= ';', 
												POS:= 0, 
												IGN:= FALSE) <> 0 THEN
							//поиск точки
							IF strTemp[i] = 46 THEN
				 				TempStrDigit := concat(TempStrDigit, '.');
							ELSE		
								TempStrDigit := concat(TempStrDigit, BYTE_TO_STRING(strTemp[i]-48)); //-48посимвольно формируем число
							end_if	
							 	
							
						ELSE
							
							gvl.DailyEnergies[n] := OSCAT_BASIC.ROUND(in:= STRING_TO_REAL(TempStrDigit), N:= 2); // из-за особенности преобразования приходиться применять функцию ROUND
							//рассчитываем индекс массива
							n := n+1;
							TempStrDigit := '';					
						END_IF											
						
					END_FOR
					
					eStateReadFile := FileWork.CLOSE;
					fFindBlock := false;	
				END_IF	
				
		END_CASE
	//
	END_IF;
	END_IF;
ELSE
	i:= i +1;
END_IF

END_PROGRAM

// Functions/CalcCRC
//Фйнкция рассчитывает конрольную сумму ModBus


FUNCTION CalcCRC : WORD
VAR_INPUT
	In:BYTE;
	
END_VAR
VAR
	i:INT;
	arrCRC: ARRAY [0..1] OF BYTE := [16#FF, 16#FF];
END_VAR

VAR CONSTANT
	srCRCHi:ARRAY[0..255] OF BYTE := [	16#00, 16#C1, 16#81, 16#40, 16#01, 16#C0, 16#80, 16#41, 16#01, 16#C0, 16#80, 16#41, 16#00, 16#C1, 16#81, 16#40, 16#01, 16#C0, 16#80, 16#41,
										16#00, 16#C1, 16#81, 16#40, 16#00, 16#C1, 16#81, 16#40, 16#01, 16#C0, 16#80, 16#41, 16#01, 16#C0, 16#80, 16#41, 16#00, 16#C1, 16#81, 16#40,
										16#00, 16#C1, 16#81, 16#40, 16#01, 16#C0, 16#80, 16#41, 16#00, 16#C1, 16#81, 16#40, 16#01, 16#C0, 16#80, 16#41, 16#01, 16#C0, 16#80, 16#41,
										16#00, 16#C1, 16#81, 16#40, 16#01, 16#C0, 16#80, 16#41, 16#00, 16#C1, 16#81, 16#40, 16#00, 16#C1, 16#81, 16#40, 16#01, 16#C0, 16#80, 16#41,
										16#00, 16#C1, 16#81, 16#40, 16#01, 16#C0, 16#80, 16#41, 16#01, 16#C0, 16#80, 16#41, 16#00, 16#C1, 16#81, 16#40, 16#00, 16#C1, 16#81, 16#40,
										16#01, 16#C0, 16#80, 16#41, 16#01, 16#C0, 16#80, 16#41, 16#00, 16#C1, 16#81, 16#40, 16#01, 16#C0, 16#80, 16#41, 16#00, 16#C1, 16#81, 16#40,
										16#00, 16#C1, 16#81, 16#40, 16#01, 16#C0, 16#80, 16#41, 16#01, 16#C0, 16#80, 16#41, 16#00, 16#C1, 16#81, 16#40, 16#00, 16#C1, 16#81, 16#40,
										16#01, 16#C0, 16#80, 16#41, 16#00, 16#C1, 16#81, 16#40, 16#01, 16#C0, 16#80, 16#41, 16#01, 16#C0, 16#80, 16#41, 16#00, 16#C1, 16#81, 16#40,
										16#00, 16#C1, 16#81, 16#40, 16#01, 16#C0, 16#80, 16#41, 16#01, 16#C0, 16#80, 16#41, 16#00, 16#C1, 16#81, 16#40, 16#01, 16#C0, 16#80, 16#41,
										16#00, 16#C1, 16#81, 16#40, 16#00, 16#C1, 16#81, 16#40, 16#01, 16#C0, 16#80, 16#41, 16#00, 16#C1, 16#81, 16#40, 16#01, 16#C0, 16#80, 16#41,
										16#01, 16#C0, 16#80, 16#41, 16#00, 16#C1, 16#81, 16#40, 16#01, 16#C0, 16#80, 16#41, 16#00, 16#C1, 16#81, 16#40, 16#00, 16#C1, 16#81, 16#40,
										16#01, 16#C0, 16#80, 16#41, 16#01, 16#C0, 16#80, 16#41, 16#00, 16#C1, 16#81, 16#40, 16#00, 16#C1, 16#81, 16#40, 16#01, 16#C0, 16#80, 16#41,
										16#00, 16#C1, 16#81, 16#40, 16#01, 16#C0, 16#80, 16#41, 16#01, 16#C0, 16#80, 16#41, 16#00, 16#C1, 16#81, 16#40];
										
	srCRCLo:ARRAY[0..255] OF BYTE := [
										16#00, 16#C0, 16#C1, 16#01, 16#C3, 16#03, 16#02, 16#C2, 16#C6, 16#06, 16#07, 16#C7, 16#05, 16#C5, 16#C4, 16#04, 16#CC, 16#0C, 16#0D, 16#CD,
										16#0F, 16#CF, 16#CE, 16#0E, 16#0A, 16#CA, 16#CB, 16#0B, 16#C9, 16#09, 16#08, 16#C8, 16#D8, 16#18, 16#19, 16#D9, 16#1B, 16#DB, 16#DA, 16#1A,
										16#1E, 16#DE, 16#DF, 16#1F, 16#DD, 16#1D, 16#1C, 16#DC, 16#14, 16#D4, 16#D5, 16#15, 16#D7, 16#17, 16#16, 16#D6, 16#D2, 16#12, 16#13, 16#D3,
										16#11, 16#D1, 16#D0, 16#10, 16#F0, 16#30, 16#31, 16#F1, 16#33, 16#F3, 16#F2, 16#32, 16#36, 16#F6, 16#F7, 16#37, 16#F5, 16#35, 16#34, 16#F4,
										16#3C, 16#FC, 16#FD, 16#3D, 16#FF, 16#3F, 16#3E, 16#FE, 16#FA, 16#3A, 16#3B, 16#FB, 16#39, 16#F9, 16#F8, 16#38, 16#28, 16#E8, 16#E9, 16#29,
										16#EB, 16#2B, 16#2A, 16#EA, 16#EE, 16#2E, 16#2F, 16#EF, 16#2D, 16#ED, 16#EC, 16#2C, 16#E4, 16#24, 16#25, 16#E5, 16#27, 16#E7, 16#E6, 16#26,
										16#22, 16#E2, 16#E3, 16#23, 16#E1, 16#21, 16#20, 16#E0, 16#A0, 16#60, 16#61, 16#A1, 16#63, 16#A3, 16#A2, 16#62, 16#66, 16#A6, 16#A7, 16#67,
										16#A5, 16#65, 16#64, 16#A4, 16#6C, 16#AC, 16#AD, 16#6D, 16#AF, 16#6F, 16#6E, 16#AE, 16#AA, 16#6A, 16#6B, 16#AB, 16#69, 16#A9, 16#A8, 16#68,
										16#78, 16#B8, 16#B9, 16#79, 16#BB, 16#7B, 16#7A, 16#BA, 16#BE, 16#7E, 16#7F, 16#BF, 16#7D, 16#BD, 16#BC, 16#7C, 16#B4, 16#74, 16#75, 16#B5,
										16#77, 16#B7, 16#B6, 16#76, 16#72, 16#B2, 16#B3, 16#73, 16#B1, 16#71, 16#70, 16#B0, 16#50, 16#90, 16#91, 16#51, 16#93, 16#53, 16#52, 16#92,
										16#96, 16#56, 16#57, 16#97, 16#55, 16#95, 16#94, 16#54, 16#9C, 16#5C, 16#5D, 16#9D, 16#5F, 16#9F, 16#9E, 16#5E, 16#5A, 16#9A, 16#9B, 16#5B,
										16#99, 16#59, 16#58, 16#98, 16#88, 16#48, 16#49, 16#89, 16#4B, 16#8B, 16#8A, 16#4A, 16#4E, 16#8E, 16#8F, 16#4F, 16#8D, 16#4D, 16#4C, 16#8C,
										16#44, 16#84, 16#85, 16#45, 16#87, 16#47, 16#46, 16#86, 16#82, 16#42, 16#43, 16#83, 16#41, 16#81, 16#80, 16#40]; 
										
	InitCRC:WORD := 16#FFFF;
END_VAR

  i:= arrCRC[1] XOR In;
  arrCRC[1]:= arrCRC[0] xor srCRCHi[i];
  arrCRC[0]:= srCRCLo[i];

  CalcCRC := SHL(arrCRC[1],8) OR  arrCRC[0];

END_FUNCTION

// Device/Application/Visualization
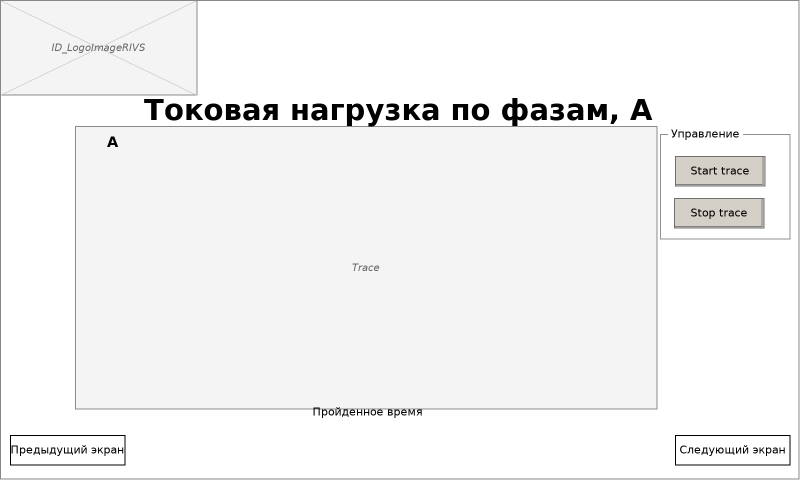
VISUALIZATION Visualization  // 800x480
VAR_IN_OUT
END_VAR
VAR
	StartTrace : BOOL;
	StopTrace : BOOL;
	bStart : BOOL;
	bStop : BOOL;
END_VAR
    Image (0,0 197x95), image: ID_LogoImageRIVS
    GroupBox (660,126 130x113), "Управление"
        Button (15,30 90x30), "Start trace"
            toggle bStart
        Button (14,72 90x30), "Stop trace"
            toggle bStop
    Trace (75,126 582x283)
        p866368322: bStart
        p3851742229: bStop
    Label (95,95 607x30), "Токовая нагрузка по фазам, А"
    Label (99,127 27x30), "A"
    Label (300,397 135x30), "Пройденное время"
    Rectangle (675,435 115x30), "Следующий экран"
        OnMouseDown:  Assign=Visualization_P, Type=Assignment
    Rectangle (10,435 115x30), "Предыдущий экран"
        OnMouseDown:  Assign=Visualization_DailyEnergies, Type=Assignment
END_VISUALIZATION

// Device/Application/Visualization_DispatchDevices
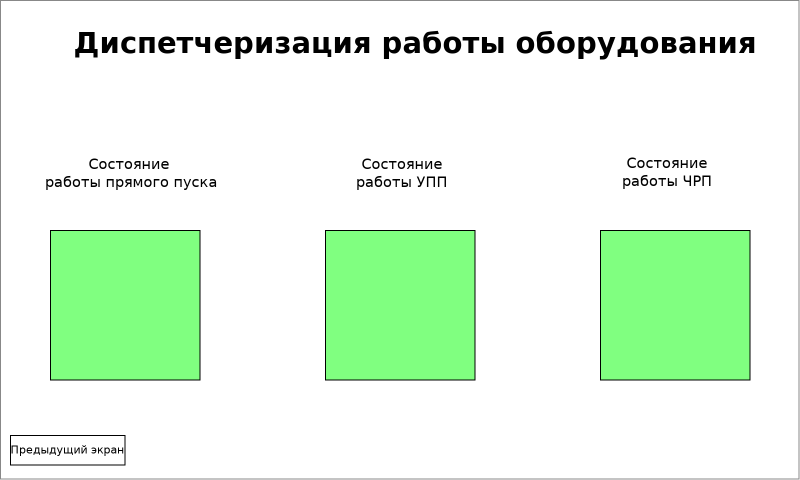
VISUALIZATION Visualization_DispatchDevices  // 800x480
    Rectangle (50,230 150x150), colour toggle: POU_DispatchDevices.DispContactor
    Rectangle (325,230 150x150), colour toggle: POU_DispatchDevices.DispUPP
    Rectangle (600,230 150x150), colour toggle: POU_DispatchDevices.DispFreqInverter
    Label (10,28 810x30), "Диспетчеризация работы оборудования"
    Label (31,148 201x50), "Состояние работы прямого пуска"
    Label (327,148 150x50), "Состояние работы УПП"
    Label (592,148 150x48), "Состояние работы ЧРП"
    Rectangle (10,435 115x30), "Предыдущий экран"
        OnMouseDown:  Assign=Visualization_P, Type=Assignment
END_VISUALIZATION

// Device/Application/Visualization_DailyEnergies
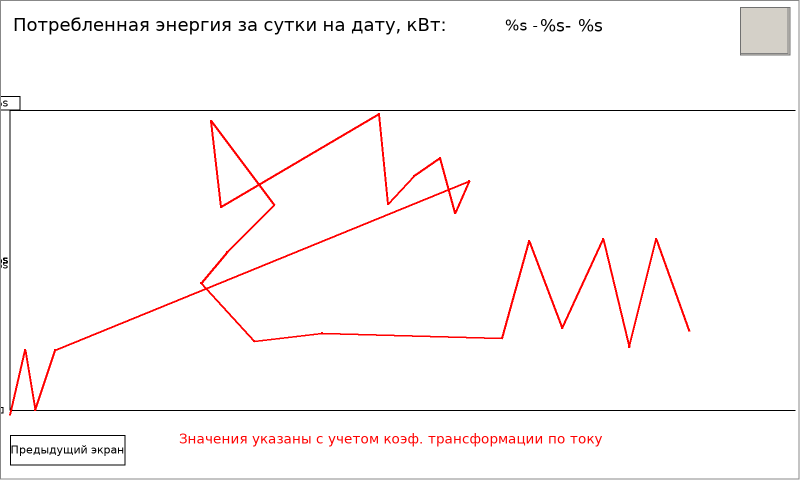
VISUALIZATION Visualization_DailyEnergies  // 800x480
    Line (10,410) (10,110)
    Line (10,410) (795,410)
    Polyline (10,415) (25,350) (35,410) (55,350) (469,181) (455,213) (440,158) (414,176) (388,204) (379,114) (221,207) (211,121) (274,205) (227,252) (201,283) (254,341) (322,333) (502,338) (529,241) (562,328) (603,239) (629,347) (656,239) (689,331)
        p1285906596: ADR(POU_VisuDailyEnergies.arrPolylineCoord)
    Rectangle (10,435 115x30), "Предыдущий экран"
        OnMouseDown:  Assign=Visualization, Type=Assignment
    Rectangle (-3,407 6x6)
        p2738717112: PLC_PRG.DotY[1]
        p3560616238: PLC_PRG.DotX[1]
    Line (0,120) (0,410), "%s", text variable: PLC_PRG.arrMetkaX[1]
        p3560616238: PLC_PRG.DotX[1]
    Label (10,10 428x30), "Потребленная энергия за сутки на дату, кВт:"
    Line (0,120) (0,400), "%s", text variable: PLC_PRG.arrMetkaX[2]
        p3560616238: PLC_PRG.DotX[2]
    Line (0,120) (0,400), "%s", text variable: PLC_PRG.arrMetkaX[3]
        p3560616238: PLC_PRG.DotX[3]
    Line (0,120) (0,400), "%s", text variable: PLC_PRG.arrMetkaX[4]
        p3560616238: PLC_PRG.DotX[4]
    Line (0,120) (0,400), "%s", text variable: PLC_PRG.arrMetkaX[5]
        p3560616238: PLC_PRG.DotX[5]
    Line (0,120) (0,400), "%s", text variable: PLC_PRG.arrMetkaX[6]
        p3560616238: PLC_PRG.DotX[6]
    Line (0,120) (0,400), "%s", text variable: PLC_PRG.arrMetkaX[7]
        p3560616238: PLC_PRG.DotX[7]
    Line (0,120) (0,400), "%s", text variable: PLC_PRG.arrMetkaX[8]
        p3560616238: PLC_PRG.DotX[8]
    Line (0,120) (0,400), "%s", text variable: PLC_PRG.arrMetkaX[9]
        p3560616238: PLC_PRG.DotX[9]
    Line (0,120) (0,400), "%s", text variable: PLC_PRG.arrMetkaX[10]
        p3560616238: PLC_PRG.DotX[10]
    Line (0,120) (0,400), "%s", text variable: PLC_PRG.arrMetkaX[11]
        p3560616238: PLC_PRG.DotX[11]
    Line (0,120) (0,400), "%s", text variable: PLC_PRG.arrMetkaX[12]
        p3560616238: PLC_PRG.DotX[12]
    Line (0,120) (0,400), "%s", text variable: PLC_PRG.arrMetkaX[13]
        p3560616238: PLC_PRG.DotX[13]
    Line (0,120) (0,400), "%s", text variable: PLC_PRG.arrMetkaX[14]
        p3560616238: PLC_PRG.DotX[14]
    Line (0,120) (0,400), "%s", text variable: PLC_PRG.arrMetkaX[15]
        p3560616238: PLC_PRG.DotX[15]
    Line (0,120) (0,400), "%s", text variable: PLC_PRG.arrMetkaX[16]
        p3560616238: PLC_PRG.DotX[16]
    Line (0,120) (0,400), "%s", text variable: PLC_PRG.arrMetkaX[17]
        p3560616238: PLC_PRG.DotX[17]
    Line (0,120) (0,400), "%s", text variable: PLC_PRG.arrMetkaX[18]
        p3560616238: PLC_PRG.DotX[18]
    Line (0,120) (0,400), "%s", text variable: PLC_PRG.arrMetkaX[19]
        p3560616238: PLC_PRG.DotX[19]
    Line (0,120) (0,400), "%s", text variable: PLC_PRG.arrMetkaX[20]
        p3560616238: PLC_PRG.DotX[20]
    Line (0,120) (0,400), "%s", text variable: PLC_PRG.arrMetkaX[21]
        p3560616238: PLC_PRG.DotX[21]
    Line (0,120) (0,400), "%s", text variable: PLC_PRG.arrMetkaX[22]
        p3560616238: PLC_PRG.DotX[22]
    Line (0,120) (0,400), "%s", text variable: PLC_PRG.arrMetkaX[23]
        p3560616238: PLC_PRG.DotX[23]
    Line (0,120) (0,400), "%s", text variable: PLC_PRG.arrMetkaX[24]
        p3560616238: PLC_PRG.DotX[24]
    Rectangle (-3,407 6x6)
        p2738717112: PLC_PRG.DotY[2]
        p3560616238: PLC_PRG.DotX[2]
    Rectangle (-3,407 6x6)
        p2738717112: PLC_PRG.DotY[3]
        p3560616238: PLC_PRG.DotX[3]
    Rectangle (-3,407 6x6)
        p2738717112: PLC_PRG.DotY[4]
        p3560616238: PLC_PRG.DotX[4]
    Rectangle (-3,407 6x6)
        p2738717112: PLC_PRG.DotY[5]
        p3560616238: PLC_PRG.DotX[5]
    Rectangle (-3,407 6x6)
        p2738717112: PLC_PRG.DotY[6]
        p3560616238: PLC_PRG.DotX[6]
    Rectangle (-3,407 6x6)
        p2738717112: PLC_PRG.DotY[7]
        p3560616238: PLC_PRG.DotX[7]
    Rectangle (-3,407 6x6)
        p2738717112: PLC_PRG.DotY[8]
        p3560616238: PLC_PRG.DotX[8]
    Rectangle (-3,407 6x6)
        p2738717112: PLC_PRG.DotY[9]
        p3560616238: PLC_PRG.DotX[9]
    Rectangle (-3,407 6x6)
        p2738717112: PLC_PRG.DotY[10]
        p3560616238: PLC_PRG.DotX[10]
    Rectangle (-3,407 6x6)
        p2738717112: PLC_PRG.DotY[11]
        p3560616238: PLC_PRG.DotX[11]
    Rectangle (-3,407 6x6)
        p2738717112: PLC_PRG.DotY[12]
        p3560616238: PLC_PRG.DotX[12]
    Rectangle (-3,407 6x6)
        p2738717112: PLC_PRG.DotY[13]
        p3560616238: PLC_PRG.DotX[13]
    Rectangle (-3,407 6x6)
        p2738717112: PLC_PRG.DotY[14]
        p3560616238: PLC_PRG.DotX[14]
    Rectangle (-3,407 6x6)
        p2738717112: PLC_PRG.DotY[15]
        p3560616238: PLC_PRG.DotX[15]
    Rectangle (-3,407 6x6)
        p2738717112: PLC_PRG.DotY[16]
        p3560616238: PLC_PRG.DotX[16]
    Rectangle (-3,407 6x6)
        p2738717112: PLC_PRG.DotY[17]
        p3560616238: PLC_PRG.DotX[17]
    Rectangle (-3,407 6x6)
        p2738717112: PLC_PRG.DotY[18]
        p3560616238: PLC_PRG.DotX[18]
    Rectangle (-3,407 6x6)
        p2738717112: PLC_PRG.DotY[19]
        p3560616238: PLC_PRG.DotX[19]
    Rectangle (-3,407 6x6)
        p2738717112: PLC_PRG.DotY[20]
        p3560616238: PLC_PRG.DotX[20]
    Rectangle (-3,407 6x6)
        p2738717112: PLC_PRG.DotY[21]
        p3560616238: PLC_PRG.DotX[21]
    Rectangle (-3,407 6x6)
        p2738717112: PLC_PRG.DotY[22]
        p3560616238: PLC_PRG.DotX[22]
    Rectangle (-3,407 6x6)
        p2738717112: PLC_PRG.DotY[23]
        p3560616238: PLC_PRG.DotX[23]
    Rectangle (-3,407 6x6)
        p2738717112: PLC_PRG.DotY[24]
        p3560616238: PLC_PRG.DotX[24]
    Rectangle (504,18 35x15), "%s -", text variable: MercuryDay
    Rectangle (538,18 35x15), "%s-", text variable: MercuryMonth
    Rectangle (573,18 35x15), "%s", text variable: MercuryYear
    Line (10,110) (795,110)
    Rectangle (-20,96 40x14), angle -45, "%s", text variable: DailyEnergies[0]
        p3560616238: PLC_PRG.XCoord[0]
    Rectangle (-20,96 40x14), angle -45, "%s", text variable: DailyEnergies[1]
        p3560616238: PLC_PRG.XCoord[1]
    Rectangle (-20,96 40x14), angle -45, "%s", text variable: DailyEnergies[2]
        p3560616238: PLC_PRG.XCoord[2]
    Rectangle (-20,96 40x14), angle -45, "%s", text variable: DailyEnergies[3]
        p3560616238: PLC_PRG.XCoord[3]
    Rectangle (-20,96 40x14), angle -45, "%s", text variable: DailyEnergies[4]
        p3560616238: PLC_PRG.XCoord[4]
    Rectangle (-20,96 40x14), angle -45, "%s", text variable: DailyEnergies[5]
        p3560616238: PLC_PRG.XCoord[5]
    Rectangle (-20,96 40x14), angle -45, "%s", text variable: DailyEnergies[6]
        p3560616238: PLC_PRG.XCoord[6]
    Rectangle (-20,96 40x14), angle -45, "%s", text variable: DailyEnergies[7]
        p3560616238: PLC_PRG.XCoord[7]
    Rectangle (-20,96 40x14), angle -45, "%s", text variable: DailyEnergies[8]
        p3560616238: PLC_PRG.XCoord[8]
    Rectangle (-20,96 40x14), angle -45, "%s", text variable: DailyEnergies[9]
        p3560616238: PLC_PRG.XCoord[9]
    Rectangle (-20,96 40x14), angle -45, "%s", text variable: DailyEnergies[10]
        p3560616238: PLC_PRG.XCoord[10]
    Rectangle (-20,96 40x14), angle -45, "%s", text variable: DailyEnergies[11]
        p3560616238: PLC_PRG.XCoord[11]
    Rectangle (-20,96 40x14), angle -45, "%s", text variable: DailyEnergies[12]
        p3560616238: PLC_PRG.XCoord[12]
    Rectangle (-20,96 40x14), angle -45, "%s", text variable: DailyEnergies[13]
        p3560616238: PLC_PRG.XCoord[13]
    Rectangle (-20,96 40x14), angle -45, "%s", text variable: DailyEnergies[14]
        p3560616238: PLC_PRG.XCoord[14]
    Rectangle (-20,96 40x14), angle -45, "%s", text variable: DailyEnergies[15]
        p3560616238: PLC_PRG.XCoord[15]
    Rectangle (-20,96 40x14), angle -45, "%s", text variable: DailyEnergies[16]
        p3560616238: PLC_PRG.XCoord[16]
    Rectangle (-20,96 40x14), angle -45, "%s", text variable: DailyEnergies[17]
        p3560616238: PLC_PRG.XCoord[17]
    Rectangle (-20,96 40x14), angle -45, "%s", text variable: DailyEnergies[18]
        p3560616238: PLC_PRG.XCoord[18]
    Rectangle (-20,96 40x14), angle -45, "%s", text variable: DailyEnergies[19]
        p3560616238: PLC_PRG.XCoord[19]
    Rectangle (-20,96 40x14), angle -45, "%s", text variable: DailyEnergies[20]
        p3560616238: PLC_PRG.XCoord[20]
    Rectangle (-20,96 40x14), angle -45, "%s", text variable: DailyEnergies[21]
        p3560616238: PLC_PRG.XCoord[21]
    Rectangle (-20,96 40x14), angle -45, "%s", text variable: DailyEnergies[22]
        p3560616238: PLC_PRG.XCoord[22]
    Rectangle (-20,96 40x14), angle -45, "%s", text variable: DailyEnergies[23]
        p3560616238: PLC_PRG.XCoord[23]
    Rectangle (-20,96 40x14), angle -45, "%s", text variable: DailyEnergies[24]
        p3560616238: PLC_PRG.XCoord[24]
    Button (740,7 50x48), image: ImagePool.setup-clipart-wrench-outline-icon-clip-art_f_85-85
        OnMouseClick:  Dialog=Visualization_ConfigDailyView, OpenModal=True, OpenCentered=True
    Label (166,429 450x20), "Значения указаны с учетом коэф. трансформации по току"
END_VISUALIZATION

// Device/Application/Visualization_P
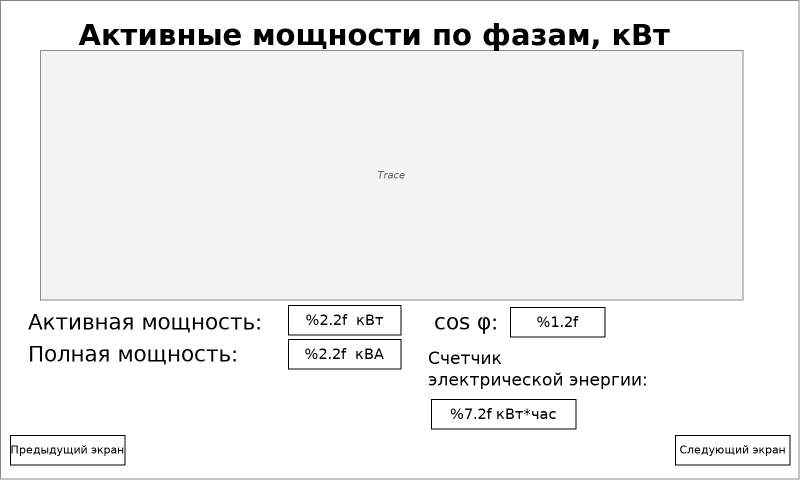
VISUALIZATION Visualization_P  // 800x480
    Trace (40,50 703x250)
    Label (24,20 701x30), "Активные мощности по фазам, кВт"
    Label (25,307 263x30), "Активная мощность:"
    Rectangle (288,305 113x30), "%2.2f кВт", text variable: POU_TracePowerActive.TraceAPowerABC
    Rectangle (10,435 115x30), "Предыдущий экран"
        OnMouseDown:  Assign=Visualization, Type=Assignment
    Label (25,339 259x30), "Полная мощность:"
    Rectangle (288,339 113x30), "%2.2f кВA", text variable: POU_TracePowerActive.TraceSPowerABC
    Rectangle (510,307 95x30), "%1.2f", text variable: PF_ABCS
    Label (421,307 90x30), "cos φ:"
    Label (425,339 242x60), "Счетчик электрической энергии:"
    Rectangle (431,399 145x30), "%7.2f кВт*час", text variable: POU_TracePowerActive.CounterPower
    Rectangle (675,435 115x30), "Следующий экран"
        OnMouseDown:  Assign=Visualization_DispatchDevices, Type=Assignment
END_VISUALIZATION

// Device/Application/Visualization_Energies
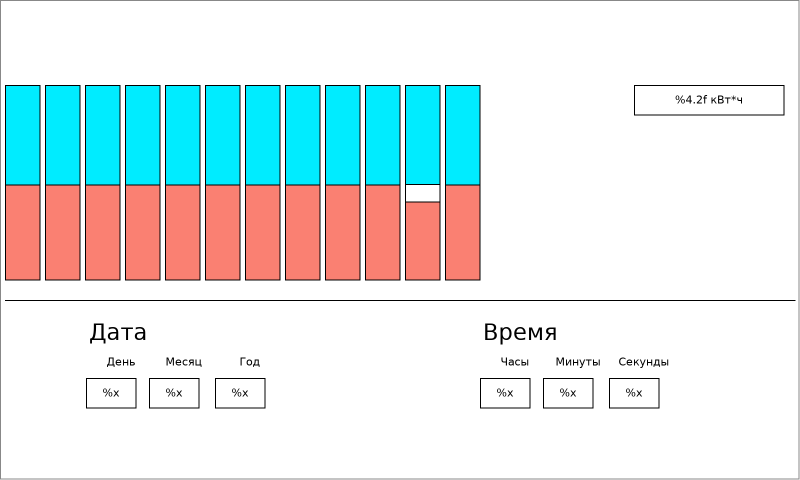
VISUALIZATION Visualization_Energies  // 800x480
    Rectangle (609,378 50x30), "%x", text variable: MercurySec
    Label (609,347 70x30), "Секунды"
    Rectangle (543,378 50x30), "%x", text variable: MercuryMin
    Label (543,347 70x30), "Минуты"
    Rectangle (480,378 50x30), "%x", text variable: MercuryHour
    Label (480,347 70x30), "Часы"
    Label (480,317 110x30), "Время"
    Rectangle (215,378 50x30), "%x", text variable: MercuryYear
    Label (215,347 70x30), "Год"
    Rectangle (149,378 50x30), "%x", text variable: MercuryMonth
    Label (149,347 70x30), "Месяц"
    Rectangle (86,378 50x30), "%x", text variable: MercuryDay
    Label (86,347 70x30), "День"
    Label (86,317 110x30), "Дата"
    Rectangle (634,85 150x30), "%4.2f кВт*ч", text variable: RealDaylyEnergyA
    Line (5,300) (795,300)
    Rectangle (5,180 35x100)
    Rectangle (5,85 35x100)
    Rectangle (45,180 35x100)
    Rectangle (45,85 35x100)
    Rectangle (85,180 35x100)
    Rectangle (85,85 35x100)
    Rectangle (125,180 35x100)
    Rectangle (125,85 35x100)
    Rectangle (165,180 35x100)
    Rectangle (165,85 35x100)
    Rectangle (205,180 35x100)
    Rectangle (205,85 35x100)
    Rectangle (245,180 35x100)
    Rectangle (245,85 35x100)
    Rectangle (285,180 35x100)
    Rectangle (285,85 35x100)
    Rectangle (325,180 35x100)
    Rectangle (325,85 35x100)
    Rectangle (365,180 35x100)
    Rectangle (365,85 35x100)
    Rectangle (405,180 35x100)
    Rectangle (405,85 35x100)
    Rectangle (445,180 35x100)
    Rectangle (445,85 35x100)
    Rectangle (405,184 35x18)
END_VISUALIZATION

// Device/Application/Visualization_EnergiesDay
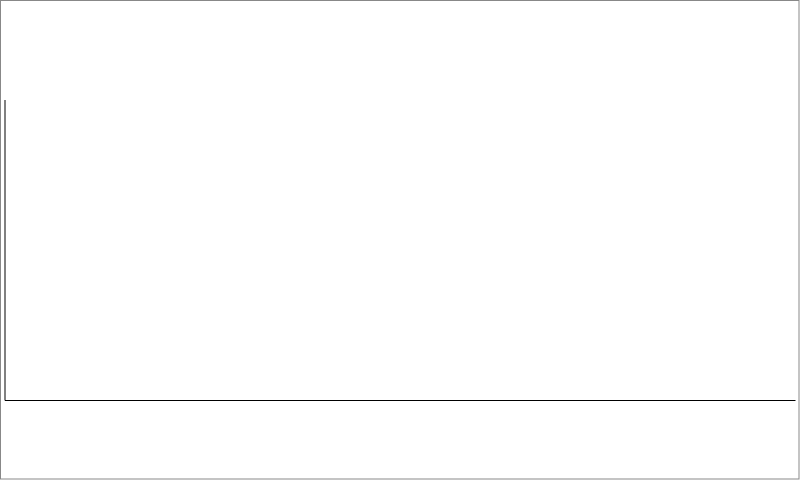
VISUALIZATION Visualization_EnergiesDay  // 800x480
    Line (5,400) (5,100)
    Line (5,400) (795,400)
END_VISUALIZATION

// Device/Application/Visualization_ConfigDailyView
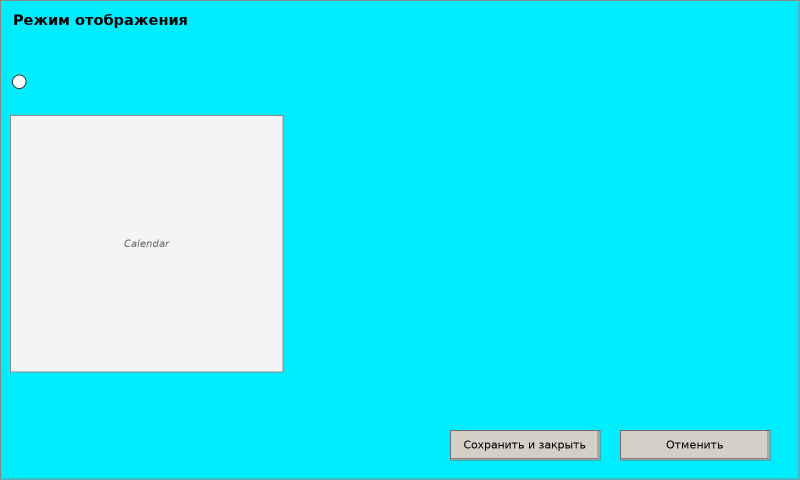
VISUALIZATION Visualization_ConfigDailyView  // 800x480
    Button (450,430 150x30), "Сохранить и закрыть"
        OnMouseClick:  Dialog=Visualization_ConfigDailyView, Result=OK, NumpadKeypadSet=True
    Button (620,430 150x30), "Отменить"
        OnMouseClick:  Dialog=Visualization_ConfigDailyView, Result=Cancel, NumpadKeypadSet=True
    RadioButton (10,49 345x65), variable: POU_VisuDailyEnergies.DailyViewConfig
        Areas[0]: Text=На текущую дату
        Areas[1]: Text=На выбранную дату
    Label (10,5 500x30), "Режим отображения"
    Calendar (10,115 273x257)
        p1438966082: POU_VisuDailyEnergies.Calender
END_VISUALIZATION

// Device/Application/Visualization_Status
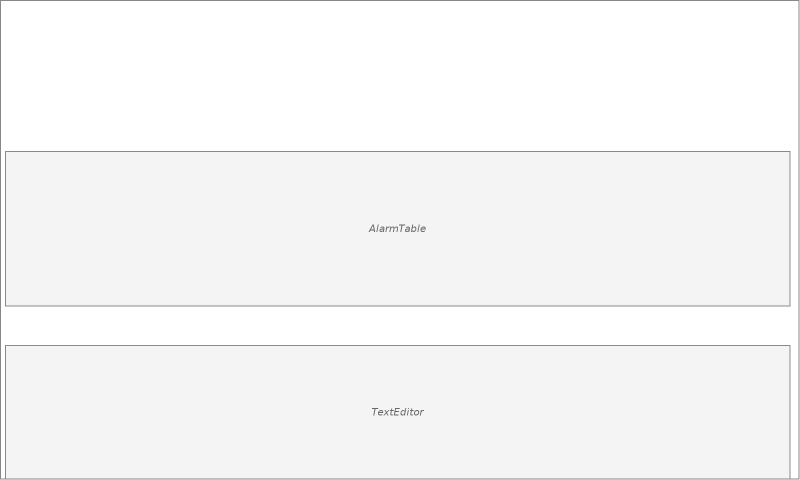
VISUALIZATION Visualization_Status  // 800x480
    TextEditor (5,345 785x134)
        p4127561890: Courier New
    AlarmTable (5,151 785x155)
        p1521930926: __All
        p1663851261: __All
END_VISUALIZATION

(* text list System (id | default)
  Apr | Apr
  April | April
  Aug | Aug
  August | August
  Dec | Dec
  December | December
  Feb | Feb
  February | February
  Fri | Fri
  Friday | Friday
  Jan | Jan
  January | January
  Jul | Jul
  July | July
  Jun | Jun
  June | June
  Mar | Mar
  March | March
  May | May
  May_3Letter | May
  Mon | Mon
  Monday | Monday
  Nov | Nov
  November | November
  Oct | Oct
  October | October
  Sat | Sat
  Saturday | Saturday
  Sep | Sep
  September | September
  Sun | Sun
  Sunday | Sunday
  Thu | Thu
  Thursday | Thursday
  Tue | Tue
  Tuesday | Tuesday
  Wed | Wed
  Wednesday | Wednesday
   |  *)

(* text list AlarmGroup (id | default)
   |  *)
